FUNCTION TimeToSeconds : LREAL
VAR_INPUT
	t : TIME;
END_VAR

TimeToSeconds := TIME_TO_LREAL(t) * 0.001;

END_FUNCTION

(* stored: Version 1.1.0.1, ProductVersion 3.1.4024.15
   POU TimeToSeconds: Id {bfe2c987-5709-0bad-0a27-ffb4c219b3a0}, SpecialFunc None *)
